FUNCTION_BLOCK SC_FirstFloor EXTENDS FB_Chain
VAR_INPUT
	bExecute : BOOL;
	bIncomingPallet : BOOL;
	bPostPalletizerRequestGranted : BOOL;
END_VAR
VAR_OUTPUT
	bPlateOpen : BOOL;
	bPalletizerRequest : BOOL;
	bSentToPostPalletizer : BOOL;
	bPostPalletizerDeliveryRequest : BOOL;
END_VAR
VAR
	fbPallChainConveyor : PalletizerConveyor;
	fbPallElevator : PalletizerElevator;
	fbPlateCyl : Cylinder;
	fbPlateLimitSen : Sensor;
	fbElevatorFrontLimit : Sensor;
	fbElevatorBackLimit : Sensor;
END_VAR

SUPER^();
bPlateOpen := fbPlateCyl.bExtended;
fbPallChainConveyor();
fbPallElevator();
fbPlateCyl();
fbPlateLimitSen();

METHOD PROTECTED   Busy : BOOL
VAR_INPUT
END_VAR

		
fbStepWorkerBusy();
CASE fbStepWorkerBusy.uiStep OF
	
	0: 
		fbPallChainConveyor.On();
		fbStepWorkerBusy
			.mAddCondition(itfStepCondition := fbElevatorBackLimit.getSignal)
			.mAddCondition(itfStepCOndition := fbElevatorFrontLimit.getSignal)
			.mNextStep(10);
			
	10: 
	
		fbPallChainConveyor.Off();
		bPalletizerRequest := FALSE;
		IF rChainController
			.releaseCheck(THIS^)
			.releaseFromChain(sChainReleasing := 'scSecondFloor', THIS^)
			.releaseResult(THIS^) 
		THEN
			fbStepWorkerBusy.mNextStep(20);
		END_IF

	20:
	
		fbPallElevator.MoveUp();
		fbStepWorkerBusy
			.mSetTimer(T#1S)
			.mNextStep(30);
			
	30:
	
		IF NOT fbPallElevator.isMoving
		THEN
			fbStepWorkerBusy
				.mSetTimer(tTime := T#2S)
				.mNextStep(40);
		END_IF
		
	40:
	
		fbPlateCyl.Extend();
		fbStepWorkerBusy
			.mSetTimer(T#2S)
			.mNextStep(45);
	
	45:	
		rChainController.releaseForChain('scSecondFloor', THIS^);	
		fbPallElevator.MoveDown();		
		fbStepWorkerBusy
			.mSetTimer(T#2S)
			.mNextStep(50);
	50:
	
		IF NOT fbPallElevator.isMoving
		THEN
			rChainController.releaseForChain('scPostPalletizer', THIS^);
			fbStepWorkerBusy.mNextStep(60);
		END_IF
	
		
	60:
	
		fbPlateCyl.Retract();
		fbStepWorkerBusy.mNextStep(100);
	
	100:
	
		IF rChainController
			.releaseCheck(THIS^)
			.releaseFromChain(sChainReleasing := 'scPostPalletizer', THIS^)
			.releaseResult(THIS^) 
		THEN

			fbPallChainConveyor.On();
			fbStepWorkerBusy.mNextStep(105);
			
		END_IF

	105:
		fbStepWorkerBusy
				.mSetTimer(T#2s)
				.mNextStep(110);
	110:		
		
		IF NOT fbElevatorBackLimit.bSignal
			AND NOT fbElevatorFrontLimit.bSignal
		THEN
		
			Done();
			fbPallChainConveyor.Off();
			fbStepWorkerBusy.mNextStep(0);
		END_IF

END_CASE
END_METHOD

METHOD PROTECTED  Error : BOOL
VAR_INPUT
END_VAR
END_METHOD

METHOD PROTECTED  Idle : BOOL
VAR_INPUT
END_VAR
END_METHOD

METHOD PROTECTED  Init : BOOL
VAR_INPUT
END_VAR
Start();
END_METHOD

METHOD PROTECTED  Prepare : BOOL
VAR_INPUT
END_VAR
END_METHOD

METHOD PROTECTED  Ready : BOOL
VAR_INPUT
END_VAR

fbStepWorkerReady();
CASE fbStepWorkerReady.uiStep OF
	
	0: 
	
		IF bExecute THEN
			fbStepWorkerReady.mNextStep(10);
		END_IF
		
	10:

		IF NOT fbElevatorFrontLimit.bSignal
			AND NOT fbElevatorBackLimit.bSignal 
		THEN
			bPalletizerRequest := TRUE;
			fbStepWorkerReady.mNextStep(20);
		END_IF
		
	20:
	
		IF bIncomingPallet
		THEN
			fbStepWorkerReady.mNextStep(0);
			Execute();
		END_IF
		
		
END_CASE
END_METHOD

METHOD PROTECTED  Waiting : BOOL
VAR_INPUT
END_VAR
END_METHOD

END_FUNCTION_BLOCK

(* stored: Version 1.1.0.1, ProductVersion 3.1.4024.2
   POU SC_FirstFloor: Id {b387d0a3-03f1-4926-83a4-5dd8702fdbd2}, SpecialFunc None
   Method Busy: Id {684ccb79-3580-4ba4-bd92-b9e29aca8ff2}
   Method Error: Id {6b3a7494-42ad-45fa-890c-59ddcc04207c}
   Method Idle: Id {c2b72847-2699-4346-84d6-e060d5196804}
   Method Init: Id {fbb5c2ac-c375-4111-a666-11fa0d41d5db}
   Method Prepare: Id {f278bc3e-762c-4932-ae86-151e2c19ccba}
   Method Ready: Id {05258b6b-2705-4ceb-9952-6379e5edf643}
   Method Waiting: Id {c7a157ad-d262-4247-b7ac-ac32cadf12cf} *)
